{attribute 'qualified_only'}
{attribute 'strict'}
{attribute 'to_string'}
TYPE TaskExecutionStates :
(
	Idle := 0,
	Running := 1,
	Done := 2,
	Error := 3
);
END_TYPE

(* stored: Version 1.1.0.1
   DUT TaskExecutionStates: Id {b5db187c-ec72-46ae-b46b-a705ba9e15fb} *)
